{attribute 'qualified_only'}
VAR_GLOBAL
	nX : INT := 0;
	nY : INT := 0;
	
	xMin : INT := -85;
	xMax : INT := 500;
	yMin : INT := -200;
	yMax : INT := 0;
END_VAR

(* stored: Version 1.1.0.1, ProductVersion 3.1.4024.12
   GVL G_Sim: Id {f59a9577-8a2e-4c4a-9fa5-4d12d7bf928a} *)
